// TIA Portal project "Contatore" (V16)

(* hardware
DEVICE "S7-1200 station_1"  S7-1200 Station
   slot 0: "Telaio di montaggio_0"  S7-1200 Rack  Rack  V1.0
   slot 1: "PLC_1"  CPU 1215C DC/DC/Rly  6ES7 215-1HG40-0XB0  V4.4
*)

// ===== PLC "PLC_1"  CPU 1215C DC/DC/Rly =====

VAR_GLOBAL   // PLC tag table "Tabella delle variabili standard"
   "Pulsante Contatore 1" AT %I1.4 : Bool;
   "Pulsante reset contatore 1" AT %I1.5 : Bool;
   "Motore in marcia n.8" AT %Q1.1 : Bool;
   "Pulsante Contatore 2" AT %I1.6 : Bool;
   "Pulsante reset contatore 2" AT %I1.7 : Bool;
   "Motore in marcia n.9" AT %Q1.2 : Bool;
   "pulsante CNT3 avanti" AT %Q1.3 : Bool;
   "pulsante CNT3 indietro" AT %Q1.4 : Bool;
   "pulsante reset cont3" AT %Q1.5 : Bool;
   "pulsante load cont3" AT %Q1.6 : Bool;
   "Motore in n.10" AT %Q1.7 : Bool;
END_VAR

// folder: System blocks/Program resources

DATA_BLOCK "Contatore 1"   // DB1
{ S7_Optimized_Access := 'TRUE' }
AUTHOR : Simatic
FAMILY : IEC
NAME : CNTR
VERSION : 1.0
// stored: InstanceOfName IEC_COUNTER
"IEC_COUNTER"
BEGIN
END_DATA_BLOCK

DATA_BLOCK "Contatore 2"   // DB2
{ S7_Optimized_Access := 'TRUE' }
AUTHOR : Simatic
FAMILY : IEC
NAME : CNTR
VERSION : 1.0
// stored: InstanceOfName IEC_COUNTER
"IEC_COUNTER"
BEGIN
END_DATA_BLOCK

DATA_BLOCK "Contatore 3"   // DB3
{ S7_Optimized_Access := 'TRUE' }
AUTHOR : Simatic
FAMILY : IEC
NAME : CNTR
VERSION : 1.0
// stored: InstanceOfName IEC_COUNTER
"IEC_COUNTER"
BEGIN
END_DATA_BLOCK

// folder: (top level)

FUNCTION "Blocco_contatori" : Void   // FC1, LAD
{ S7_Optimized_Access := 'TRUE' }
VERSION : 0.1
BEGIN

REGION Network 1
   // Conteggio avanti
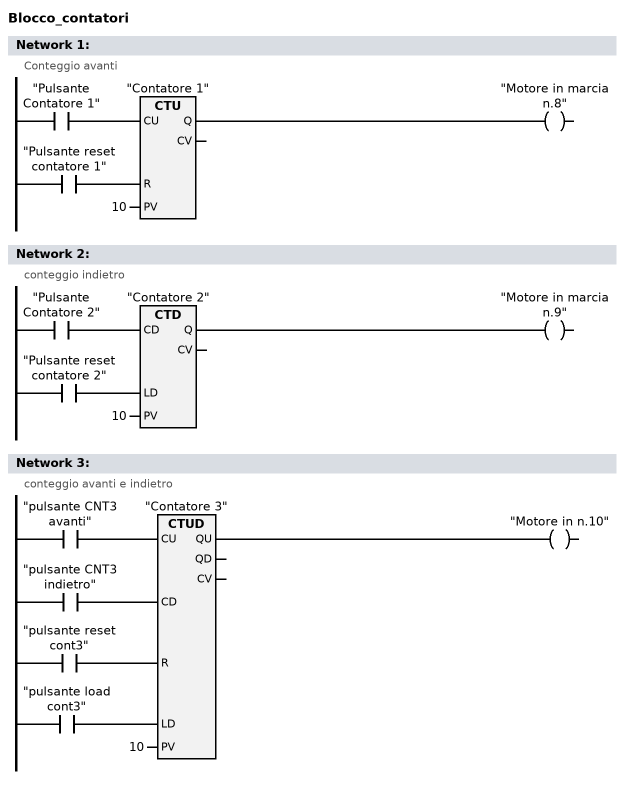
   "Contatore 1".CTU(CU := "Pulsante Contatore 1", R := "Pulsante reset contatore 1", PV := 10);
   "Motore in marcia n.8" := "Contatore 1".Q;
END_REGION

REGION Network 2
   // conteggio indietro
   "Contatore 2".CTD(CD := "Pulsante Contatore 2", LD := "Pulsante reset contatore 2", PV := 10);
   "Motore in marcia n.9" := "Contatore 2".Q;
END_REGION

REGION Network 3
   // conteggio avanti e indietro
   "Contatore 3".CTUD(CU := "pulsante CNT3 avanti",
                      CD := "pulsante CNT3 indietro",
                      R := "pulsante reset cont3",
                      LD := "pulsante load cont3",
                      PV := 10);
   "Motore in n.10" := "Contatore 3".QU;
END_REGION
END_FUNCTION

ORGANIZATION_BLOCK "Main"   // OB1, LAD, ProgramCycle
TITLE = "Main Program Sweep (Cycle)"
{ S7_Optimized_Access := 'TRUE' }
VERSION : 0.1
   VAR_INPUT
      Initial_Call : Bool;   // Initial call of this OB
      Remanence : Bool;   // =True, if remanent data are available
   END_VAR
BEGIN

REGION Network 1
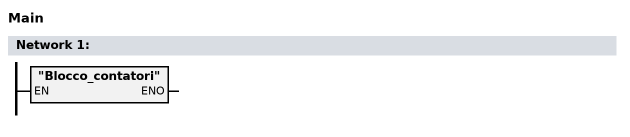
   RUNG wire#powerrail
      "Blocco_contatori"()
   END_RUNG
   // the same network as SCL:
   "Blocco_contatori"();
END_REGION
END_ORGANIZATION_BLOCK